(* Logix 5000 project; controller Marker_Machine_with_Secuencers Emulate 5570 rev 30.12; software revision 30.01 *)

TASK T00 (continuous, watchdog 500 ms) : P00_Marker

MODULES
   Local : Emulate 5570 (ICP 2, rev 30.12)
      Inputs_Outputs : vendor 1 type 0 code 15 (ICP 3, rev 1.1, Output RPI 50 ms)
           Local:3:O.Data[0].0   // Motor Forward
           Local:3:O.Data[0].1   // Stop Motor
           Local:3:O.Data[0].2   // Motor reverse
           Local:3:O.Data[0].3   // Cylinder Up
           Local:3:O.Data[0].4   // Pipe Cylinder
END_MODULES

VAR_GLOBAL   (* controller tags *)
   Automatic_Manual : BOOL;   // Automatic 0 Manual 1
   cylinder_up : DINT;
   cylinder_up_sensor : BOOL;   // cylinder up = 1 cylinder down = 0
   e_stop : BOOL;
   home : BOOL;
   initial_conditions : BOOL;
   LH_Overtravel : BOOL;
   marker_ready : BOOL;
   Motor_Forward : BOOL;
   Motor_Reverse : DINT;
   Motor_Stop : DINT;
   PB_Reset : BOOL;
   PB_Start : BOOL;
   pipe_loaded : BOOL;
   Pipe_press : BOOL;
   Position_1 : BOOL;
   Position_2 : BOOL;
   Position_3 : BOOL;
   RH_Overtravel : BOOL;
   Secuencer : DINT;
   T4 : TIMER[25] := ([0].PRE := 250, [1].PRE := 250, [2].PRE := 250);
END_VAR

PROGRAM P00_Marker   (* main routine R00_MainRoutine *)

ROUTINE R00_MainRoutine   (* ladder *)
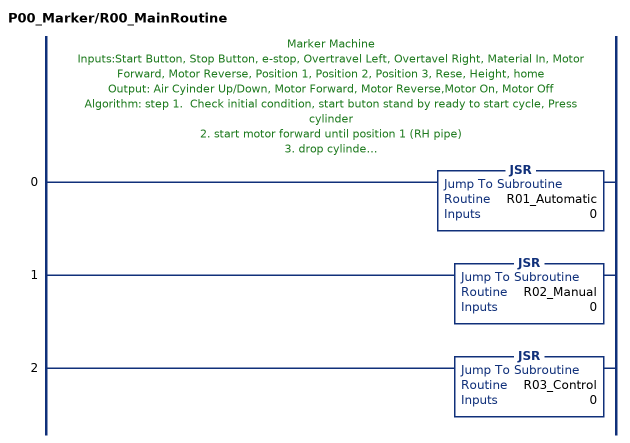
   // Marker Machine
   // Inputs:Start Button, Stop Button, e-stop, Overtravel Left, Overtavel Right, Material In, Motor Forward, Motor Reverse, Position 1, Position 2, Position 3, Rese, Height, home
   // Output: Air Cyinder Up/Down, Motor Forward, Motor Reverse,Motor On, Motor Off
   // Algorithm: step 1.  Check initial condition, start buton stand by ready to start cycle, Press cylinder
   // 2. start motor forward until position 1 (RH pipe)
   // 3. drop cylinder
   // 4. Initiate sequence marker ready marker up
   // 5. marker up Return marker to position 2
   // 6. drop cylinder
   // 7.  Initiate sequence marker ready marker up
   // 8. marker up Return marker to position 1
   // 6. drop cylinder
   // 9.  Initiate sequence marker ready marker up
   // 10.marker up Return marker to home
   // 11. Look for home
   // 12 release press cylinder
   0: JSR(R01_Automatic,0);
   1: JSR(R02_Manual,0);
   2: JSR(R03_Control,0);
END_ROUTINE

ROUTINE R01_Automatic   (* ladder *)
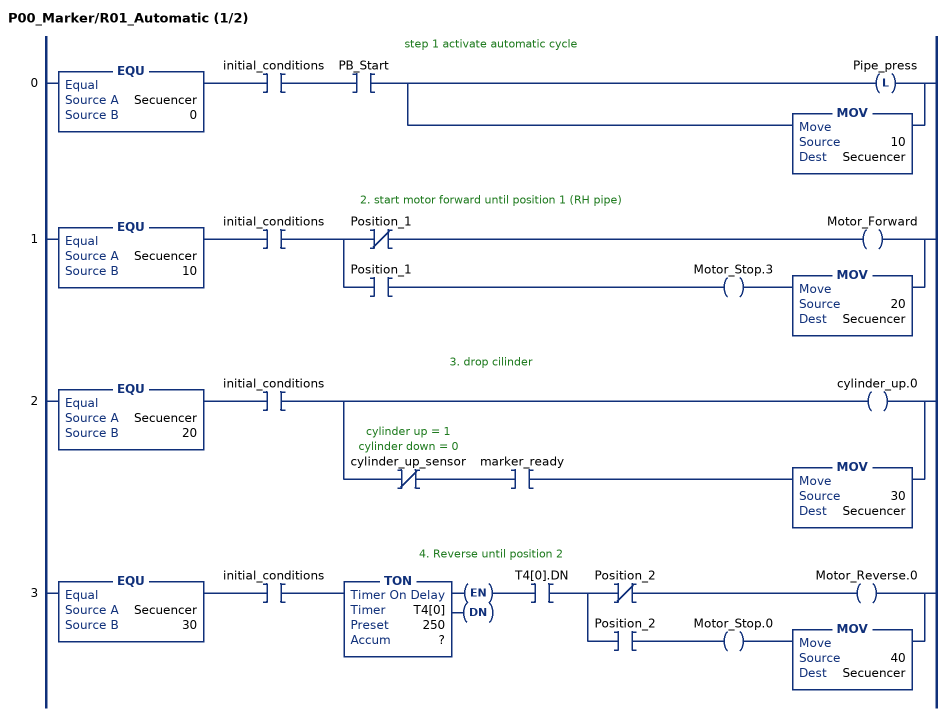
   // step 1 activate automatic cycle
   0: EQU(Secuencer,0)XIC(initial_conditions)XIC(PB_Start)[OTL(Pipe_press) ,MOV(10,Secuencer) ];
   // 2. start motor forward until position 1 (RH pipe)
   1: EQU(Secuencer,10)XIC(initial_conditions)[XIO(Position_1) OTE(Motor_Forward) ,XIC(Position_1) OTE(Motor_Stop.3) MOV(20,Secuencer) ];
   // 3. drop cilinder
   2: EQU(Secuencer,20)XIC(initial_conditions)[OTE(cylinder_up.0) ,XIO(cylinder_up_sensor) XIC(marker_ready) MOV(30,Secuencer) ];
   // 4. Reverse until position 2
   3: EQU(Secuencer,30)XIC(initial_conditions)TON(T4[0],?,?)XIC(T4[0].DN)[XIO(Position_2) OTE(Motor_Reverse.0) ,XIC(Position_2) OTE(Motor_Stop.0) MOV(40,Secuencer) ];
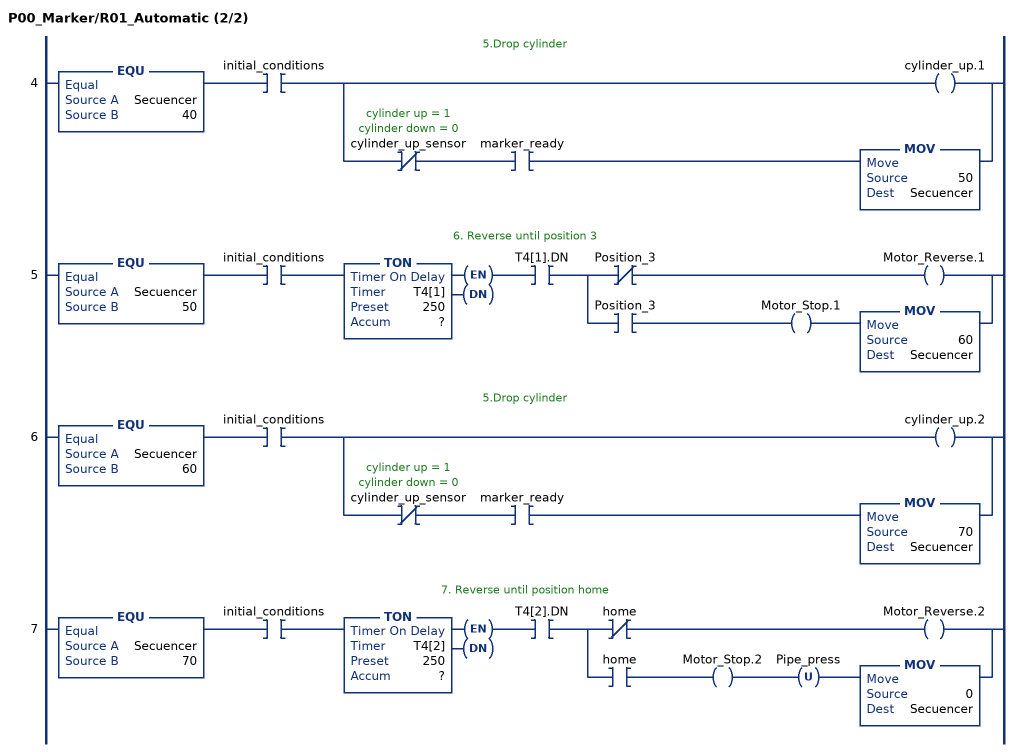
   // 5.Drop cylinder
   4: EQU(Secuencer,40)XIC(initial_conditions)[OTE(cylinder_up.1) ,XIO(cylinder_up_sensor) XIC(marker_ready) MOV(50,Secuencer) ];
   // 6. Reverse until position 3
   5: EQU(Secuencer,50)XIC(initial_conditions)TON(T4[1],?,?)XIC(T4[1].DN)[XIO(Position_3) OTE(Motor_Reverse.1) ,XIC(Position_3) OTE(Motor_Stop.1) MOV(60,Secuencer) ];
   // 5.Drop cylinder
   6: EQU(Secuencer,60)XIC(initial_conditions)[OTE(cylinder_up.2) ,XIO(cylinder_up_sensor) XIC(marker_ready) MOV(70,Secuencer) ];
   // 7. Reverse until position home
   7: EQU(Secuencer,70)XIC(initial_conditions)TON(T4[2],?,?)XIC(T4[2].DN)[XIO(home) OTE(Motor_Reverse.2) ,XIC(home) OTE(Motor_Stop.2) OTU(Pipe_press) MOV(0,Secuencer) ];
END_ROUTINE

ROUTINE R02_Manual   (* ladder *)
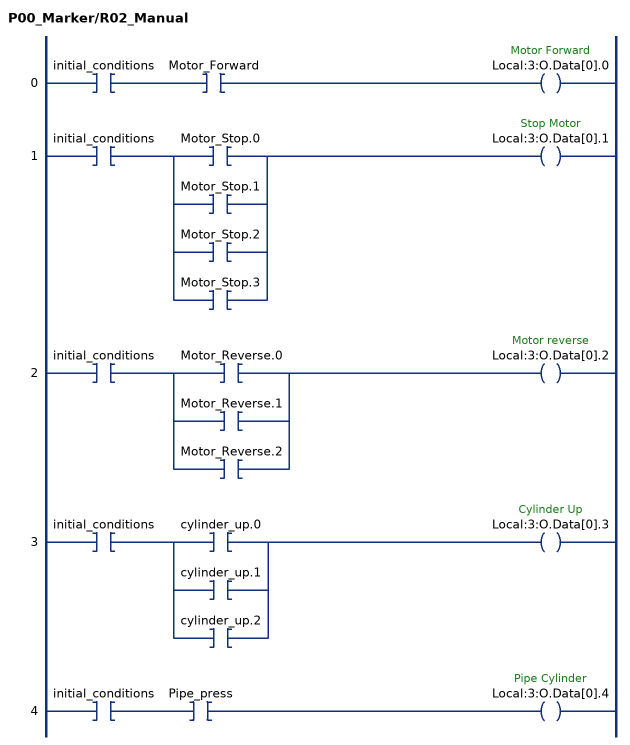
   0: XIC(initial_conditions)XIC(Motor_Forward)OTE(Local:3:O.Data[0].0);
   1: XIC(initial_conditions)[XIC(Motor_Stop.0) ,XIC(Motor_Stop.1) ,XIC(Motor_Stop.2) ,XIC(Motor_Stop.3) ]OTE(Local:3:O.Data[0].1);
   2: XIC(initial_conditions)[XIC(Motor_Reverse.0) ,XIC(Motor_Reverse.1) ,XIC(Motor_Reverse.2) ]OTE(Local:3:O.Data[0].2);
   3: XIC(initial_conditions)[XIC(cylinder_up.0) ,XIC(cylinder_up.1) ,XIC(cylinder_up.2) ]OTE(Local:3:O.Data[0].3);
   4: XIC(initial_conditions)XIC(Pipe_press)OTE(Local:3:O.Data[0].4);
END_ROUTINE

ROUTINE R03_Control   (* ladder *)
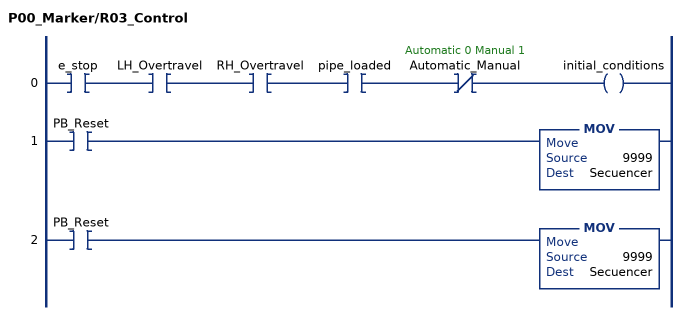
   0: XIC(e_stop)XIC(LH_Overtravel)XIC(RH_Overtravel)XIC(pipe_loaded)XIO(Automatic_Manual)OTE(initial_conditions);
   1: XIC(PB_Reset)MOV(9999,Secuencer);
   2: XIC(PB_Reset)MOV(9999,Secuencer);
END_ROUTINE
END_PROGRAM
